FUNCTION_BLOCK motor_vfd
VAR_INPUT
	//Run Feedback from Motor Starter
	run_feedback : BOOL; 
	//Reset trigger for Runtime Maint
	runtime_maint_reset : BOOL;
	//Run Request from PLC Program
	run_request : BOOL;
	//Requested Speed From PLC Program
	speed_request : REAL;
	//Speed Feedback from VFD
	speed_feedback : REAL;
	//VFD is Faulted
	fault : BOOL;
	//Daily Reset from GENERAL POU
	daily_reset : BOOL;
END_VAR
VAR_OUTPUT
	//Tells the motor to start when true, stop when false
	run_command : BOOL;
	//VFD Fault Alarm
	runtime_today : REAL;
	//Accumulated Runtime Hours Today
	runtime_total : REAL;
	//Resettable Runtime for Maintenance purposes, Description is user adjustable
	runtime_maint : REAL;
	//Speed Command to VFD
	speed_command : REAL;
	//Motor Status(Calculated) 0=Off, 1=Running, 2=Faulted
	status : INT;
END_VAR
VAR
	//Runtime Timer Tags, 1 Minute Timer
	runtime_ton : TON;
	runtime_pt : TIME := T#1M;
	runtime_et : TIME;
	//Runtime Today Counter
	runtime_today_ctu : CTU;
	runtime_today_ctu_pv : WORD;
	runtime_today_ctu_cv : REAL;
	//Total Runtime Minute Counter
	runtime_total_minute_ctu : CTU;
	runtime_total_minute_ctu_reset : BOOL;
	runtime_total_minute_ctu_pv : WORD :=60;
	runtime_total_minute_ctu_cv : REAL;
	//Total Runtime Hour Counter
	runtime_total_hour_ctu : CTU;
	runtime_total_hour_ctu_reset : BOOL;
	runtime_total_hour_ctu_pv : WORD;
	//Maintenance Runtime Minute Counter
	runtime_maint_minute_ctu : CTU;
	runtime_maint_minute_ctu_reset : BOOL;
	runtime_maint_minute_ctu_pv : WORD :=60;
	runtime_maint_minute_ctu_cv : REAL;
	//Maintenance Runtime Hour Counter
	runtime_maint_hour_ctu : CTU;
	runtime_maint_hour_ctu_pv : WORD;
END_VAR
VAR // added by the converter: edge detectors and wires of the graphical bodies
    _w1, _w2, _w3, _w4, _w5 : BOOL;
END_VAR

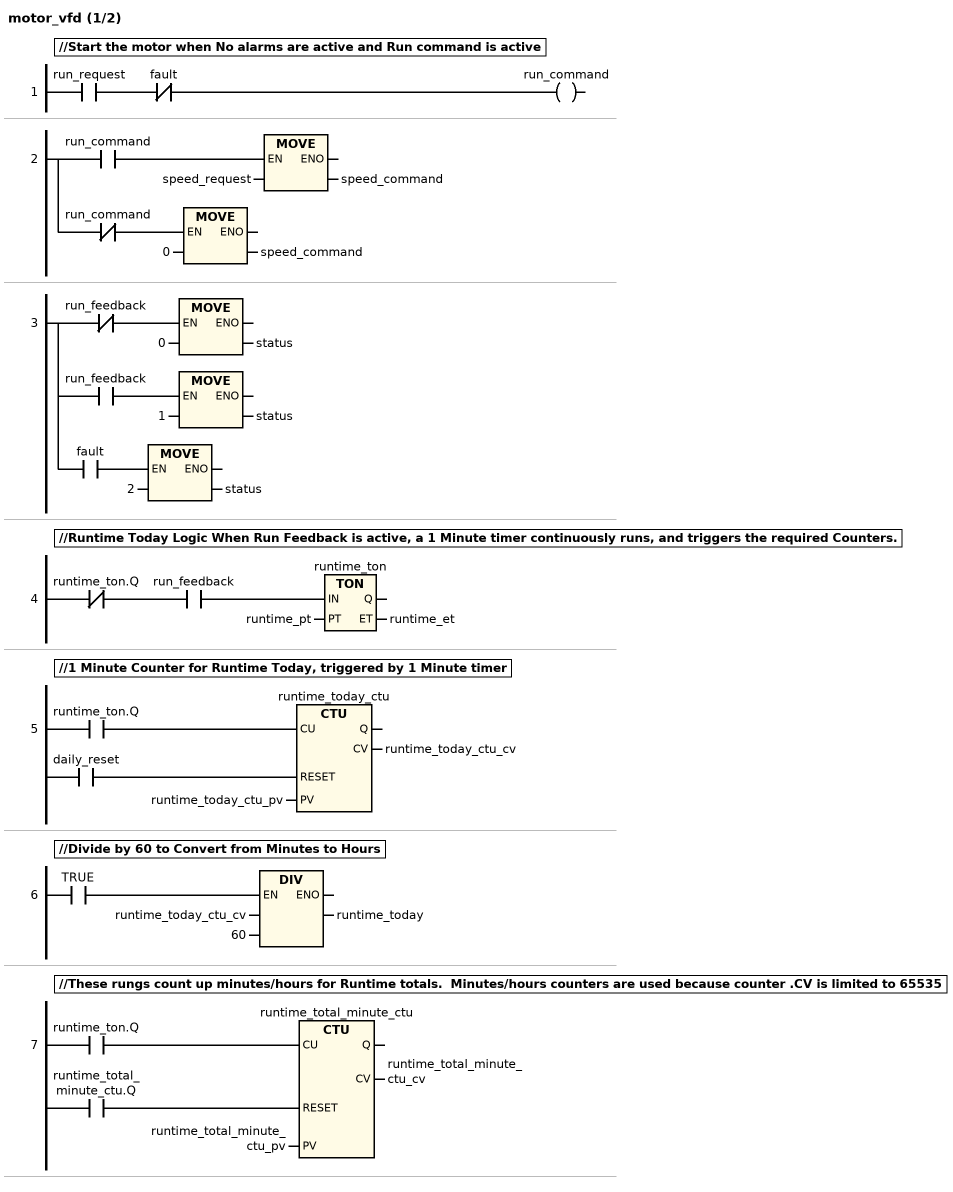
// NETWORK 1
// label: //Start the motor when No alarms are active and Run command is active
run_command := run_request AND NOT fault;

// NETWORK 2
_w1 := run_command;
IF _w1 THEN speed_command := speed_request; END_IF
_w2 := NOT run_command;
IF _w2 THEN speed_command := 0; END_IF
(* _w1 OR _w2; result not used *)

// NETWORK 3
_w3 := NOT run_feedback;
IF _w3 THEN status := 0; END_IF
_w4 := run_feedback;
IF _w4 THEN status := 1; END_IF
_w5 := fault;
IF _w5 THEN status := 2; END_IF
(* _w3 OR _w4 OR _w5; result not used *)

// NETWORK 4
// label: //Runtime Today Logic When Run Feedback is active, a 1 Minute timer continuously runs, and triggers the required Counters.
runtime_ton(IN := NOT runtime_ton.Q AND run_feedback, PT := runtime_pt, ET => runtime_et); // TON

// NETWORK 5
// label: //1 Minute Counter for Runtime Today, triggered by 1 Minute timer
runtime_today_ctu(
    CU := runtime_ton.Q,
    RESET := daily_reset,
    PV := runtime_today_ctu_pv,
    CV => runtime_today_ctu_cv); // CTU

// NETWORK 6
// label: //Divide by 60 to Convert from Minutes to Hours
runtime_today := runtime_today_ctu_cv / 60;

// NETWORK 7
// label: //These rungs count up minutes/hours for Runtime totals.  Minutes/hours counters are used because counter .CV is limited to 65535
runtime_total_minute_ctu(
    CU := runtime_ton.Q,
    RESET := runtime_total_minute_ctu.Q,
    PV := runtime_total_minute_ctu_pv,
    CV => runtime_total_minute_ctu_cv); // CTU

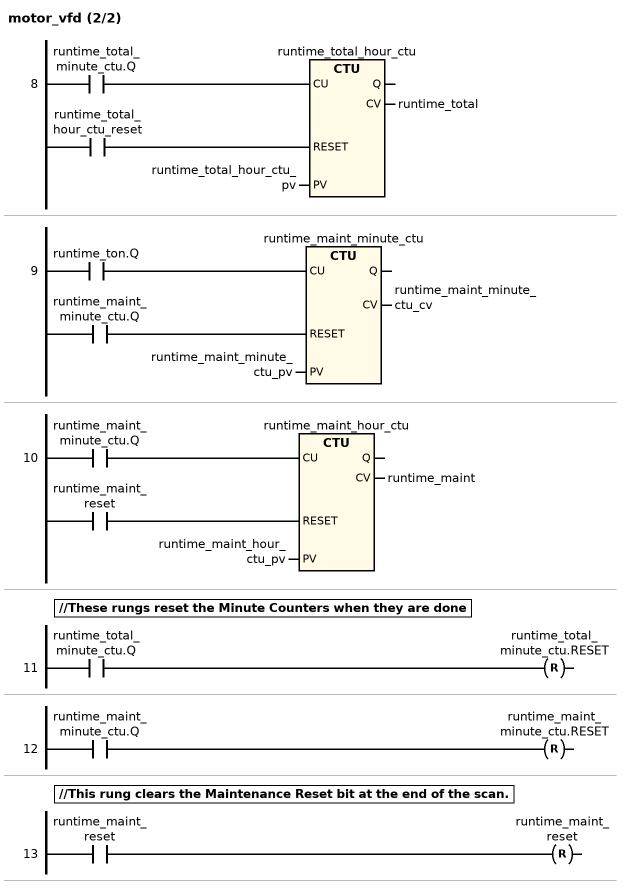
// NETWORK 8
runtime_total_hour_ctu(
    CU := runtime_total_minute_ctu.Q,
    RESET := runtime_total_hour_ctu_reset,
    PV := runtime_total_hour_ctu_pv,
    CV => runtime_total); // CTU

// NETWORK 9
runtime_maint_minute_ctu(
    CU := runtime_ton.Q,
    RESET := runtime_maint_minute_ctu.Q,
    PV := runtime_maint_minute_ctu_pv,
    CV => runtime_maint_minute_ctu_cv); // CTU

// NETWORK 10
runtime_maint_hour_ctu(
    CU := runtime_maint_minute_ctu.Q,
    RESET := runtime_maint_reset,
    PV := runtime_maint_hour_ctu_pv,
    CV => runtime_maint); // CTU

// NETWORK 11
// label: //These rungs reset the Minute Counters when they are done
runtime_total_minute_ctu.RESET R= runtime_total_minute_ctu.Q;

// NETWORK 12
runtime_maint_minute_ctu.RESET R= runtime_maint_minute_ctu.Q;

// NETWORK 13
// label: //This rung clears the Maintenance Reset bit at the end of the scan.
runtime_maint_reset R= runtime_maint_reset;

END_FUNCTION_BLOCK

(* stored: Version 1.1.0.1, ProductVersion 3.1.4024.12
   POU motor_vfd: Id {60a210a4-48dd-4db3-b672-c8198b95c310}, SpecialFunc None *)
